INTERFACE I_ioInterface

METHOD getOutputs
VAR_IN_OUT
	stSimOut : ST_inputs_analog;
END_VAR
END_METHOD

METHOD setInputs
VAR_INPUT
	stValvePos	: ST_ValvePos;
	eCraneState : E_CraneStatus;
END_VAR
END_METHOD

END_INTERFACE

(* stored: Version 1.1.0.1
   Itf I_ioInterface: Id {505e22f3-9238-449c-bbd1-997bbf60e9b5}
   Method getOutputs: Id {769e2e60-e724-4929-93fb-c1aacf6fa0f0}
   Method setInputs: Id {56972086-c862-4a68-a44a-8dbc05c607fc} *)
